FUNCTION_BLOCK SS3_ifb_Bunker_ps (* Composite FB wrapping other FBs *)
  (* Standard: 61499-2 *)
  (* Version 1.0, 2025-05-16, PS_Transformer_for_Unknown *)
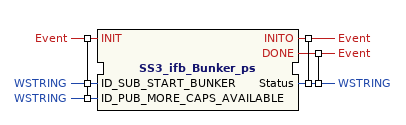
  EVENT_INPUT
    INIT WITH ID_SUB_START_BUNKER, ID_PUB_MORE_CAPS_AVAILABLE; (* Initialization Request *)
  END_EVENT
  EVENT_OUTPUT
    INITO WITH Status; (* Initialization Confirm *)
    DONE WITH Status; (* Execution Confirmation *)
  END_EVENT
  VAR_INPUT
    ID_SUB_START_BUNKER : WSTRING;
    ID_PUB_MORE_CAPS_AVAILABLE : WSTRING;
  END_VAR
  VAR_OUTPUT
    Status : WSTRING; (* Output event qualifier *)
  END_VAR
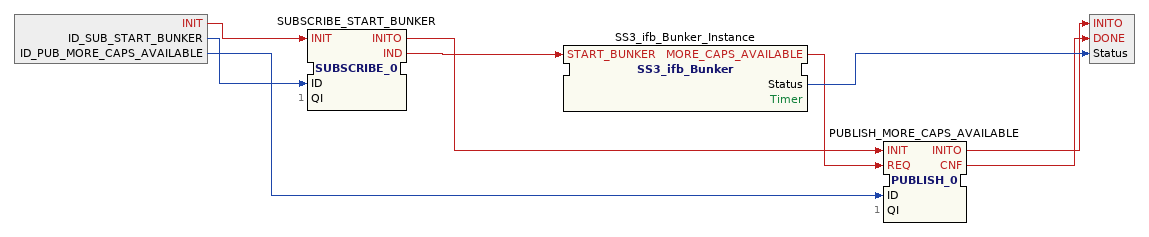
  FBS
    SS3_ifb_Bunker_Instance : SS3_ifb_Bunker;
    SUBSCRIBE_START_BUNKER : SUBSCRIBE_0(QI := 1);
    PUBLISH_MORE_CAPS_AVAILABLE : PUBLISH_0(QI := 1);
  END_FBS
  EVENT_CONNECTIONS
    INIT TO SUBSCRIBE_START_BUNKER.INIT;
    SUBSCRIBE_START_BUNKER.INITO TO PUBLISH_MORE_CAPS_AVAILABLE.INIT;
    PUBLISH_MORE_CAPS_AVAILABLE.INITO TO INITO;
    SUBSCRIBE_START_BUNKER.IND TO SS3_ifb_Bunker_Instance.START_BUNKER;
    SS3_ifb_Bunker_Instance.MORE_CAPS_AVAILABLE TO PUBLISH_MORE_CAPS_AVAILABLE.REQ;
    PUBLISH_MORE_CAPS_AVAILABLE.CNF TO DONE;
  END_CONNECTIONS
  DATA_CONNECTIONS
    ID_SUB_START_BUNKER TO SUBSCRIBE_START_BUNKER.ID;
    ID_PUB_MORE_CAPS_AVAILABLE TO PUBLISH_MORE_CAPS_AVAILABLE.ID;
    SS3_ifb_Bunker_Instance.Status TO Status;
  END_CONNECTIONS
END_FUNCTION_BLOCK
